TYPE ST_ClampingPositionConfig :
STRUCT
    fReadyPosition : LREAL;
    fApproachPosition : LREAL;
    fClampPosition : LREAL;
END_STRUCT
END_TYPE

(* stored: Version 1.1.0.1, ProductVersion 3.1.4026.20
   DUT ST_ClampingPositionConfig: Id {4deac8e7-13c7-4405-ad7b-9dd23e3b8863} *)
